{attribute 'GeneratedUsingTerminal: EL6201-0000-0017'}
{attribute addProperty BoxType "EL6201-0000-0017"}
{attribute addProperty Id "Slave_19A_DI0BOOL1Slave_19A_DI1BOOL1Slave_19A_DI2BOOL1Slave_19A_DI3BOOL1Slave_19B_DI0BOOL1Slave_19B_DI1BOOL1Slave_19B_DI2BOOL1Slave_19B_DI3BOOL1"}
{attribute addProperty CRC "1416018293"}
{attribute addProperty Size "8"}
TYPE Slave_19_Inputs_5466B975 :
STRUCT
	{attribute addProperty Name "Slave_19A_DI0"}
	Slave_19A_DI0 : BOOL;
	{attribute addProperty Name "Slave_19A_DI1"}
	Slave_19A_DI1 : BOOL;
	{attribute addProperty Name "Slave_19A_DI2"}
	Slave_19A_DI2 : BOOL;
	{attribute addProperty Name "Slave_19A_DI3"}
	Slave_19A_DI3 : BOOL;
	{attribute addProperty Name "Slave_19B_DI0"}
	Slave_19B_DI0 : BOOL;
	{attribute addProperty Name "Slave_19B_DI1"}
	Slave_19B_DI1 : BOOL;
	{attribute addProperty Name "Slave_19B_DI2"}
	Slave_19B_DI2 : BOOL;
	{attribute addProperty Name "Slave_19B_DI3"}
	Slave_19B_DI3 : BOOL;
END_STRUCT
END_TYPE

(* stored: Version 1.2.0.0, ProductVersion 3.1.4024.9
   DUT Slave_19_Inputs_5466B975: Id {e0e7722a-8748-4435-ae75-0a850c41d020} *)
